{attribute 'qualified_only'}
{attribute 'strict'}
TYPE E_ReadCSVStep :
(
	Step_Init := 0,
	Step_Open	:= 10,	
	Step_OpenWaite		:= 20,
	Step_ReadSingleLine		:= 30,
	Step_ReadSingleLineWait	,
	Step_ParseSingleLine,
	Step_Close	,
	Step_ErrorOrEnd		:= 999
);
END_TYPE

(* stored: Version 1.1.0.1, ProductVersion 3.1.4022.16
   DUT E_ReadCSVStep: Id {204ef1e6-0cae-48b7-b7e0-f77d599e2358} *)
